// TIA Portal project "Carroponte" (V15.1)

(* hardware
DEVICE "S71500/ET200MP station_1"  S7-1500 station
   slot 0: "Telaio di montaggio_0"  Rack  6ES7 590-1***0-0AA0
   slot 1: "PLC_1"  CPU 1516-3 PN/DP  6ES7 516-3AN01-0AB0  V2.5
      slot 3: "Display CPU_1"  6ES7591-1BA00-0AA0
   slot 2: "DI 32x24VDC HF_1"  DI 32x24VDC HF  6ES7 521-1BL00-0AB0  V2.1
   slot 3: "DQ 32x24VDC/0.5A HF_1"  DQ 32x24VDC/0.5A HF  6ES7 522-1BL01-0AB0  V1.0
   slot 4: "AI 8xU/I/RTD/TC ST_1"  AI 8xU/I/RTD/TC ST  6ES7 531-7KF00-0AB0  V2.1
   slot 5: "AQ 4xU/I ST_1"  AQ 4xU/I ST  6ES7 532-5HD00-0AB0  V2.1
*)

// ===== PLC "PLC_1"  CPU 1516-3 PN/DP =====

VAR_GLOBAL   // PLC tag table "Tabella delle variabili_1"
   "motore_sale" AT %Q0.0 : Bool;
   "motore_scende" AT %Q0.1 : Bool;
   "motore_indietro" AT %Q0.2 : Bool;
   "motore_avanti" AT %Q0.3 : Bool;
   "motore_sx" AT %Q0.4 : Bool;
   "motore_dx" AT %Q0.5 : Bool;
   "emergenza" AT %I0.0 : Bool;
   "manuale" AT %I0.1 : Bool;
   "indietro" AT %I0.3 : Bool;
   "avanti" AT %I0.2 : Bool;
   "destra" AT %I0.4 : Bool;
   "sinistra" AT %I0.5 : Bool;
   "scende" AT %I0.6 : Bool;
   "sale" AT %I0.7 : Bool;
   "automatico" AT %I1.0 : Bool;
   "inizializzazione" AT %I1.1 : Bool;
   "avvio" AT %I1.2 : Bool;
   "stop" AT %I1.3 : Bool;
   "prossimiti" AT %I1.4 : Bool;
   "T1" AT %I1.5 : Bool;
   "T2" AT %I1.6 : Bool;
   "S1" AT %I2.0 : Bool;
   "S2" AT %I2.1 : Bool;
   "S3" AT %I2.2 : Bool;
END_VAR

DATA_BLOCK "DB_comandi"   // DB1
{ S7_Optimized_Access := 'FALSE' }
VERSION : 0.1
   VAR
      bypassEmergenza : Bool := true;
      emergenza : Bool;
      manuale : Bool;
      indietro : Bool;
      avanti : Bool;
      destra : Bool;
      sinistra : Bool;
      scende : Bool;
      sale : Bool;
      eseguiAutomatico : Bool;
      automatico : Bool;
      inizializzazione : Bool;
      avvio : Bool;
      stop : Bool;
      prossimiti : Bool;
      t1 : Bool;
      t2 : Bool;
      s1 : Bool;
      s2 : Bool;
      s3 : Bool;
   END_VAR
BEGIN
END_DATA_BLOCK

DATA_BLOCK "DB_stati"   // DB2
{ S7_Optimized_Access := 'FALSE' }
VERSION : 0.1
   VAR
      fineCorsaSalita : Bool;
      sale : Bool;
      scende : Bool;
      avanti : Bool;
      indietro : Bool;
      sinistra : Bool;
      destra : Bool;
      fineCorsaX : Bool;
      fineCorsaY : Bool;
      inizioCorsaX : Bool;
      inizioCorsaY : Bool;
      movimentoX : Bool;
      movimentoY : Bool;
      movimento : Bool;
      partenzaConosciuta : Bool;
   END_VAR
BEGIN
END_DATA_BLOCK

DATA_BLOCK "DB_posizioni"   // DB3
{ S7_Optimized_Access := 'FALSE' }
VERSION : 0.1
   VAR
      "A" : Bool;   // Posizione 1
      "B" : Bool;   // Posizione 2
      C : Bool;   // Posizione 3
      D : Bool;   // Posizione 4
      "E" : Bool;   // Posizione 5
      F : Bool;   // Posizione 6
      destinazione : UInt := 6;   // Numero corrispondente alla lettera
      posizione : UInt;   // posizione in cui mi trovo
      Sconosciuto : Bool;   // Caso base carroponte
   END_VAR
BEGIN
END_DATA_BLOCK

FUNCTION "FC_uscite" : Void   // FC1, SCL
{ S7_Optimized_Access := 'TRUE' }
VERSION : 0.1
BEGIN
   IF NOT "DB_comandi".emergenza OR "DB_comandi".bypassEmergenza THEN
       "motore_avanti" := "DB_stati".avanti;
       "motore_indietro" := "DB_stati".indietro;
       "motore_dx" := "DB_stati".destra;
       "motore_sx" := "DB_stati".sinistra;
       "motore_sale" := "DB_stati".sale;
       "motore_scende" := "DB_stati".scende;
   END_IF;
END_FUNCTION

FUNCTION "FC_ingressi" : Void   // FC2, SCL
{ S7_Optimized_Access := 'TRUE' }
VERSION : 0.1
BEGIN
   //imposto gli ingressi sul DB
   "DB_comandi".emergenza := "emergenza";
   "DB_comandi".manuale := "manuale";
   "DB_comandi".automatico := "automatico";

   IF "DB_comandi".manuale THEN
       "DB_comandi".indietro := "indietro";
       "DB_comandi".avanti := "avanti";
       "DB_comandi".destra := "destra";
       "DB_comandi".sinistra := "sinistra";
       "DB_comandi".scende := "scende";
       "DB_comandi".sale := "sale";
   END_IF;

   "DB_comandi".inizializzazione := "inizializzazione";
   "DB_comandi".avvio := "avvio";
   "DB_comandi".stop := "stop";

   "DB_comandi".eseguiAutomatico := (
       "DB_comandi".automatico AND
       "DB_comandi".avvio
   ) OR "DB_comandi".eseguiAutomatico;

   IF "DB_comandi".stop THEN
       "DB_comandi".eseguiAutomatico := FALSE;
   END_IF;

   "DB_comandi".prossimiti := "prossimiti";
   "DB_comandi".t1 := "T1";
   "DB_comandi".t2 := "T2";
   "DB_comandi".s1 := "S1";
   "DB_comandi".s2 := "S2";
   "DB_comandi".s3 := "S3";


   "DB_comandi".manuale := "DB_comandi".manuale AND NOT "DB_comandi".automatico;
   "DB_comandi".automatico := "DB_comandi".automatico AND NOT "DB_comandi".manuale;

   //imposto le uscite sul DB
   IF NOT "DB_comandi".automatico THEN

       "DB_stati".sale := "sale";
       "DB_stati".scende := "scende";
       "DB_stati".indietro := "indietro";
       "DB_stati".avanti := "avanti";
       "DB_stati".sinistra := "sinistra";
       "DB_stati".destra := "destra";

   END_IF;

   "DB_stati".fineCorsaX := "T2";
   "DB_stati".inizioCorsaX := "T1";
   "DB_stati".fineCorsaY := "S1";
   "DB_stati".inizioCorsaY := "S3";
   "DB_stati".fineCorsaSalita := "prossimiti";


   "DB_stati".movimentoX := "DB_stati".destra OR "DB_stati".sinistra;
   "DB_stati".movimentoY := "DB_stati".avanti OR "DB_stati".indietro;
   "DB_stati".movimento := "DB_stati".movimentoX OR "DB_stati".movimentoY;

   "DB_posizioni".A := "DB_stati".fineCorsaX AND "DB_stati".fineCorsaY;
   "DB_posizioni".B := "DB_stati".inizioCorsaX AND "DB_stati".fineCorsaY;
   "DB_posizioni".C := "DB_stati".fineCorsaX AND "DB_comandi".s2;
   "DB_posizioni".D := "DB_stati".inizioCorsaX AND "DB_comandi".s2;
   "DB_posizioni".E := "DB_stati".fineCorsaX AND "DB_stati".inizioCorsaY;
   "DB_posizioni".F := "DB_stati".inizioCorsaX AND "DB_stati".inizioCorsaY;

   "DB_posizioni".Sconosciuto := NOT (
       "DB_posizioni".A OR
       "DB_posizioni".B OR
       "DB_posizioni".C OR
       "DB_posizioni".D OR
       "DB_posizioni".E OR
       "DB_posizioni".F
       );

   IF "DB_posizioni".A THEN
       "DB_posizioni".posizione := 1;
   ELSIF "DB_posizioni".B THEN
       "DB_posizioni".posizione := 2;
   ELSIF "DB_posizioni".C THEN
       "DB_posizioni".posizione := 3;
   ELSIF "DB_posizioni".D THEN
       "DB_posizioni".posizione := 4;
   ELSIF "DB_posizioni".E THEN
       "DB_posizioni".posizione := 5;
   ELSIF "DB_posizioni".F THEN
       "DB_posizioni".posizione := 6;
   ELSE
       "DB_posizioni".posizione := 0;
   END_IF;

   IF ("DB_comandi".avvio) THEN
       "DB_stati".partenzaConosciuta := FALSE;
   END_IF;
END_FUNCTION

FUNCTION "FC_manuale" : Void   // FC3, SCL
{ S7_Optimized_Access := 'TRUE' }
VERSION : 0.1
BEGIN
   IF ("DB_comandi".manuale OR "DB_comandi".bypassEmergenza) AND (NOT "DB_comandi".automatico) THEN

       IF "DB_comandi".indietro THEN
           "DB_stati".indietro := TRUE;
           "DB_stati".avanti := FALSE;
       END_IF;

       IF "DB_comandi".avanti THEN
           "DB_stati".avanti := TRUE;
           "DB_stati".indietro := FALSE;
       END_IF;

       IF "DB_comandi".destra THEN
           "DB_stati".destra := TRUE;
           "DB_stati".sinistra := FALSE;
       END_IF;

       IF "DB_comandi".sinistra THEN
           "DB_stati".sinistra := TRUE;
           "DB_stati".destra := FALSE;
       END_IF;

       IF "DB_comandi".sale THEN
           "DB_stati".sale := TRUE;
           "DB_stati".scende := FALSE;
       END_IF;

       IF "DB_comandi".scende THEN
           "DB_stati".scende := TRUE;
           "DB_stati".sale := FALSE;
       END_IF;

   END_IF;
END_FUNCTION

FUNCTION "FC_sicurezza" : Void   // FC4, SCL
{ S7_Optimized_Access := 'TRUE' }
VERSION : 0.1
BEGIN
   //fine corsa
   //
   IF "DB_comandi".manuale OR ("DB_posizioni".posizione = "DB_posizioni".destinazione) THEN
       "DB_comandi".eseguiAutomatico := FALSE;
   END_IF;

   IF "DB_stati".inizioCorsaY THEN
       "DB_stati".indietro := FALSE;
   END_IF;

   IF "DB_stati".fineCorsaY THEN
       "DB_stati".avanti := FALSE;
   END_IF;

   IF "DB_stati".inizioCorsaX THEN
       "DB_stati".sinistra := FALSE;
   END_IF;

   IF "DB_stati".fineCorsaX THEN
       "DB_stati".destra := FALSE;
   END_IF;

   IF "DB_stati".fineCorsaSalita THEN
       "DB_stati".sale := FALSE;
   END_IF;

   IF "DB_stati".movimentoX AND "DB_stati".movimentoY THEN
       "DB_stati".avanti := FALSE;
       "DB_stati".indietro := FALSE;
       "DB_stati".destra := FALSE;
       "DB_stati".sinistra := FALSE;
       "DB_stati".sale := FALSE;
       "DB_stati".scende := FALSE;
   END_IF;

   IF "DB_stati".movimentoX OR "DB_stati".movimentoY THEN
       "DB_stati".sale := FALSE;
       "DB_stati".scende := FALSE;
   END_IF;

   IF "DB_comandi".stop THEN
       "DB_comandi".eseguiAutomatico := FALSE;
       "DB_stati".avanti := FALSE;
       "DB_stati".indietro := FALSE;
       "DB_stati".destra := FALSE;
       "DB_stati".sinistra := FALSE;
       "DB_stati".sale := FALSE;
       "DB_stati".scende := FALSE;
   END_IF;
END_FUNCTION

FUNCTION "FC_automatico" : Void   // FC5, SCL
{ S7_Optimized_Access := 'TRUE' }
VERSION : 0.1
BEGIN
   IF "DB_comandi".automatico AND "DB_comandi".eseguiAutomatico AND NOT "DB_comandi".manuale THEN
       IF "DB_comandi".inizializzazione THEN
           "DB_posizioni".destinazione := 1;
       END_IF;

       IF NOT ("DB_posizioni".posizione = "DB_posizioni".destinazione)
       THEN
           IF "DB_posizioni".Sconosciuto AND NOT "DB_stati".partenzaConosciuta
           THEN
               IF NOT "DB_stati".fineCorsaX AND NOT "DB_stati".movimentoY
               THEN
                   "DB_stati".destra := TRUE;
               ELSE
                   "DB_stati".avanti := TRUE;
               END_IF;
           END_IF;

           IF NOT "DB_posizioni".Sconosciuto
           THEN
               "DB_stati".partenzaConosciuta := TRUE;
           END_IF;

           IF "DB_stati".partenzaConosciuta AND NOT ("DB_posizioni".destinazione = "DB_posizioni".posizione)
           THEN
               IF NOT "DB_posizioni".Sconosciuto THEN
                   "DB_stati".avanti := "DB_stati".indietro := FALSE;
                   "DB_stati".sinistra := "DB_stati".destra := FALSE;

                   IF (NOT ("DB_stati".avanti OR "DB_stati".indietro)) AND NOT (("DB_posizioni".posizione MOD 2 = "DB_posizioni".destinazione MOD 2))
                   THEN
                       IF NOT "DB_stati".fineCorsaX AND (("DB_posizioni".posizione MOD 2 = 0) AND (NOT ("DB_posizioni".destinazione MOD 2 = 0)))
                       THEN
                           "DB_stati".destra := TRUE;
                       ELSIF NOT "DB_stati".inizioCorsaX AND ((NOT ("DB_posizioni".posizione MOD 2 = 0)) AND ("DB_posizioni".destinazione MOD 2 = 0))
                       THEN
                           "DB_stati".sinistra := TRUE;
                       END_IF;
                   END_IF;

                   IF (NOT ("DB_stati".sinistra OR "DB_stati".destra))
                   THEN
                       IF "DB_posizioni".posizione > "DB_posizioni".destinazione
                       THEN
                           "DB_stati".avanti := TRUE;
                       ELSIF "DB_posizioni".posizione < "DB_posizioni".destinazione
                       THEN
                           "DB_stati".indietro := TRUE;
                       END_IF;
                   END_IF;

               END_IF;
           END_IF;
       END_IF;
       IF ("DB_posizioni".destinazione = "DB_posizioni".posizione) THEN
           "DB_stati".avanti := "DB_stati".indietro := FALSE;
           "DB_stati".sinistra := "DB_stati".destra := FALSE;
       END_IF;
   END_IF;
END_FUNCTION

ORGANIZATION_BLOCK "Main"   // OB1, LAD, ProgramCycle
TITLE = "Main Program Sweep (Cycle)"
{ S7_Optimized_Access := 'TRUE' }
VERSION : 0.1
   VAR_INPUT
      Initial_Call : Bool;   // Initial call of this OB
      Remanence : Bool;   // =True, if remanent data are available
   END_VAR
   VAR_TEMP   // added for the SCL form of the ladder/FBD networks
      _w1 : Bool;
      _w2 : Bool;
      _w3 : Bool;
      _w4 : Bool;
   END_VAR
BEGIN

REGION Network 1
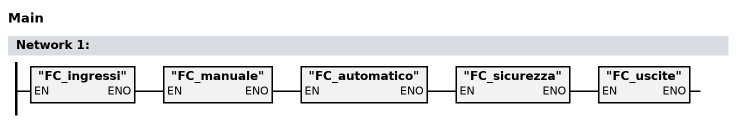
   RUNG wire#powerrail
      "FC_ingressi"()
      "FC_manuale"()
      "FC_automatico"()
      "FC_sicurezza"()
      "FC_uscite"()
   END_RUNG
   // the same network as SCL:
   "FC_ingressi"(ENO => #_w1);
   "FC_manuale"(EN := #_w1, ENO => #_w2);
   "FC_automatico"(EN := #_w2, ENO => #_w3);
   "FC_sicurezza"(EN := #_w3, ENO => #_w4);
   IF #_w4 THEN "FC_uscite"(); END_IF;
END_REGION
END_ORGANIZATION_BLOCK